(* PLC project  *)

PROGRAM P
  VAR  (* added by the conversion: wires and edge detectors of the diagram *)
    _AND3_OUT : BOOL;
  END_VAR

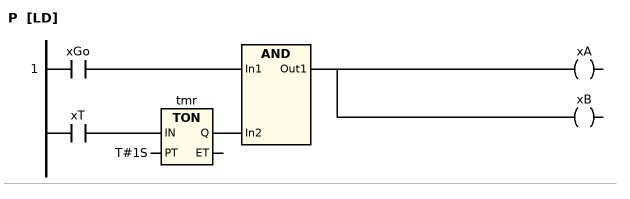
(* LD diagram, written out as Structured Text *)
tmr(IN := xT, PT := T#1S);
_AND3_OUT := xGo AND tmr.Q;
xA := _AND3_OUT;
xB := _AND3_OUT;
END_PROGRAM
